FUNCTION_BLOCK SC_PrePalletizer EXTENDS FB_Chain
VAR_INPUT
	bPalletizerRequest : BOOL;
	bExecute : BOOL;
END_VAR
VAR_OUTPUT
	bSentToPalletizer : BOOL;
	bPalletAvailable : BOOL;
END_VAR
VAR
	fbRollConvEntrance : RollerConveyor;
	fbRollConvPrePallet : RollerConveyor;
	fbPalletAvailable : Sensor;
END_VAR

SUPER^();
bPalletAvailable := fbPalletAvailable.bSignal;

METHOD PROTECTED   Busy : BOOL
VAR_INPUT
END_VAR
fbStepWorkerBusy();
CASE fbStepWorkerBusy.uiStep OF
	
	0: 
		fbRollConvEntrance.On();
		fbRollConvPrePallet.On();
		IF NOT bPalletAvailable
		THEN
			bSentToPalletizer := TRUE;
			fbStepWorkerReady.mNextStep(10);
		END_IF

	10:
		IF NOT bPalletizerRequest
		THEN
		
			bSentToPalletizer := FALSE;
			fbRollConvPrePallet.Off();
			fbStepWorkerReady.mNextStep(0);
			
			Done();
			
		ELSIF bPalletAvailable
		THEN
			fbRollConvEntrance.Off();
		END_IF
		
END_CASE
END_METHOD

METHOD PROTECTED  Error : BOOL
VAR_INPUT
END_VAR
END_METHOD

METHOD PROTECTED  Idle : BOOL
VAR_INPUT
END_VAR
END_METHOD

METHOD PROTECTED  Init : BOOL
VAR_INPUT
END_VAR
Start();
END_METHOD

METHOD PROTECTED  Prepare : BOOL
VAR_INPUT
END_VAR
END_METHOD

METHOD PROTECTED  Ready : BOOL
VAR_INPUT
END_VAR

fbStepWorkerReady();
CASE fbStepWorkerReady.uiStep OF
	
	0:
		IF bExecute
		THEN
			fbStepWorkerReady.mNextStep(5);
		END_IF
		
	5: 
		IF NOT bPalletAvailable
		THEN
			fbRollConvEntrance.On();
		ELSIF bPalletAvailable
		THEN
			fbRollConvEntrance.Off();
			fbStepWorkerReady.mNextStep(10);
		END_IF
		
	10:
		IF bPalletizerRequest
		THEN
			fbStepWorkerReady.mNextStep(0);
			Execute();
		END_IF
		
END_CASE
END_METHOD

METHOD PROTECTED  Waiting : BOOL
VAR_INPUT
END_VAR
END_METHOD

END_FUNCTION_BLOCK

(* stored: Version 1.1.0.1, ProductVersion 3.1.4024.2
   POU SC_PrePalletizer: Id {5dff49bc-e989-4c97-b519-5d232efdac58}, SpecialFunc None
   Method Busy: Id {b4960330-9bf6-4d42-8bb8-1d990e9bb531}
   Method Error: Id {b6393260-4a97-48b4-9678-ce4cc88b9229}
   Method Idle: Id {54eba9a7-05d0-49e7-ae84-357a62c152ff}
   Method Init: Id {c1ac30ae-7cbf-4b3c-8c5e-e45fdf7336c2}
   Method Prepare: Id {a3187a60-cfef-4867-a914-8a22f27efc5b}
   Method Ready: Id {f386c72d-a0bb-42a7-afcd-096615a8b827}
   Method Waiting: Id {8c3351a7-4525-4e7c-b2e7-a30d64b5a1c4} *)
